// SIMATIC S7-200 project (STEP 7-Micro/WIN), CPU 222 REL 02.01

SYMBOL_TABLE USER1
P1_STOP          I0.0     // ARRESTO DEL NASTRO DAL POSTO 1
P2_STOP          I0.1     // ARRESTO DEL NASTRO DAL POSTO 2
P1_DX            I0.2     // AVVIO DEL NASTRO IN AUTOMATICO DAL POSTO 1 VERSO DX
P2_DX            I0.3     // AVVIO DEL NASTRO IN AUTOMATICO DAL POSTO 2 VERSO DX
P1_SX            I0.4     // AVVIO DEL NASTRO IN AUTOMATICO DAL POSTO 1 VERSO SX
P2_SX            I0.5     // AVVIO DEL NASTRO IN AUTOMATICO DAL POSTO 2 VERSO SX
B1_DX            I0.6     // AVVIO DEL NASTRO IN MODO INTERMITTENTE VERSO DX
B2_DX            I0.7     // AVVIO DEL NASTRO IN MODO INTERMITTENTE VERSO DX
B1               I1.0     // RELE' FOTOELETTRICO ON COMMUTAZIONE BUIO
B2               I1.1     // RELE' FOTOELETTRICO ON COMMUTAZIONE BUIO
DX_AUTO          M0.0     // START AUTOMATICO VERSO DESTRA
SX_AUTO          M0.1     // START AUTOMATICO VERSO SINISTRA
MOT_DX           Q0.0     // MOVIMENTO NASTRO VERSO DESTRA
MOT_SX           Q0.1     // MOVIMENTO NASTRO VERSO SINISTRA
RIT_AVV_DX       T37      // RITARDO INTENZIONALE AVVIAMENTO AUTO VERSO DX
RIT_AVV_SX       T38      // RITARDO INTENZIONALE AVVIAMENTO AUTO VERSO SX
END_SYMBOL_TABLE

ORGANIZATION_BLOCK MAIN:OB1
TITLE=DPS 207 NASTRO TRASPORTATORE
BEGIN
Network 1 // COMANDO AUTOMATICO MOTORE VERSO DESTRA
// IL MOVIMENTO AUTOMATICO VERSO DESTRA AVVIENE:
// - AZIONE SUL PULSANTE P1_DX
// - AZIONE SUL PULSANTE P2_DX
// - ATTESA DI 1,5 SECONDI
// IL MOVIMENTO AUTOMATICO VERSO DESTRA SI ARRESTA:
// - AZIONE PULSANTE P1_STOP
// - AZIONE PULSANTE P2_STOP
// - INTERVENTO RELE' FOTELETTRICO  B2 = ON  ( FINECORSA DESTRA)  
// - SE VIENE COMANDATO IL MOVIMENTO VERSO SINISTRA IN AUTOMATICO  SX_AUTO = ON
// - SE NON VIENE ATTTIVATO IL COMANDO INTERMITTENTE B1_DX = ON O B2_DX = ON
LD     P1_DX:I0.2
O      P2_DX:I0.3
LD     DX_AUTO:M0.0
AN     B1_DX:I0.6
AN     B2_DX:I0.7
OLD
AN     P1_STOP:I0.0
AN     P2_STOP:I0.1
LPS
AN     B2:I1.1
AN     SX_AUTO:M0.1
=      DX_AUTO:M0.0
LPP
TON    RIT_AVV_DX:T37, 15
Network 2 // COMANDO INTERMITTENTE VERSO DESTRA
// IL MOVIMENTO INTERMITTENTE VERSO DESTRA AVVIENE:
// - CONTESTUALMENTE ALLA PRESSIONE DEI PULSANTI B1_DX O B2_DX
// - FINO ALL'INTERVENTO DEL RELE' FOTOELETTRICO B2= ON   ( FINECORSA DESTRA)  
LD     RIT_AVV_DX:T37
O      B1_DX:I0.6
O      B2_DX:I0.7
AN     B2:I1.1
=      MOT_DX:Q0.0
Network 3 // COMANDO AUTOMATICO MOTORE VERSO SINISTRA
// IL MOVIMENTO AUTOMATICO VERSO SINISTRA AVVIENE:
// - AZIONE SUL PULSANTE P1_SX
// - AZIONE SUL PULSANTE P2_SX
// - ATTESA DI 1,5 SECONDI
// IL MOVIMENTO AUTOMATICO VERSO SINISTRA SI ARRESTA:
// - AZIONE PULSANTE P1_STOP
// - AZIONE PULSANTE P2_STOP
// - INTERVENTO RELE' FOTELETTRICO  B1 = ON  ( FINECORSA SINISTRA)  
// - SE VIENE COMANDATO IL MOVIMENTO VERSO DESTRA IN AUTOMATICO  DX_AUTO = ON
// - SE NON VIENE ATTIVATO IL COMANDO INTERMITTENTE B1_DX = ON O B2_DX = ON
LD     P1_SX:I0.4
O      P2_SX:I0.5
O      SX_AUTO:M0.1
AN     P1_STOP:I0.0
AN     P2_STOP:I0.1
LPS
AN     B1:I1.0
LPS
A      RIT_AVV_SX:T38
AN     DX_AUTO:M0.0
=      MOT_SX:Q0.1
LPP
AN     B1_DX:I0.6
AN     B2_DX:I0.7
=      SX_AUTO:M0.1
LPP
TON    RIT_AVV_SX:T38, 15
END_ORGANIZATION_BLOCK
